(* Logix 5000 project; controller PBS_Perfusion vendor 1 type 14 code 217 rev 32.14; software revision 32.03; part 10 of 27 *)
(* tags used below, declared in another part *)
   Cfg_HasOper : BOOL;   // 1=Operator (unlocked) exists, can be selected
   Cfg_HasOperLocked : BOOL;   // 1=Operator Locked exists, can be selected
   Cfg_HasProg : BOOL;   // 1=Program (unlocked) exists, can be selected
   Cfg_HasProgLocked : BOOL;   // 1=Program Locked exists, can be selected
   Cfg_HasExt : BOOL;   // 1=External exists, can be selected
   Cfg_HasMaint : BOOL;   // 1=Maintenance exists, can be selected
   Cfg_HasMOoS : BOOL;   // 1=Maintenance Out of Service exists, can be selected
   Cfg_OvrdOverLock : BOOL;   // 1=Override supersedes Prog/Oper Lock, 0=don't override Lock
   Cfg_ExtOverLock : BOOL;   // 1=External supersedes Prog/Oper Lock, 0=don't override Lock
   Cfg_ProgNormal : BOOL;   // Normal Source: 1=Program if no requests; 0=Operator if no requests
   Cfg_PCmdPriority : BOOL;   // Command Priority: 1=Program Cmds Win; 0=Operator Cmds Win
   Cfg_PCmdProgAsLevel : BOOL;   // 1=PCmd_Prog used as a Level (1=Prog, 0=Oper)
   Cfg_PCmdLockAsLevel : BOOL;   // 1=PCmd_Lock used as a Level (1=Lock, 0=Unlock)
   Cfg_ExtAcqAsLevel : BOOL;   // 1=XCmd_Acq used as Level (1=Acq, 0=Rel)
   MCmd_Acq : BOOL;   // Maintenance Command to Acquire (Oper/Prog/Ovrd to Maint)
   OCmd_Oper : BOOL;   // Operator Command to select Operator (Prog to Oper)
   OCmd_Prog : BOOL;   // Operator Command to select Program (Oper to Prog)
   OCmd_Lock : BOOL;   // Operator Command to Lock Operator (disallow Program)
   Sts_eSrc : INT;   // Selection enum: .8=Ext, .7=OoS, .6=Oper, .5=Prog, .4=Ovrd, .3=Maint, .2=Hand, .1=Norm, .0=Lock
   Sts_bSrc : INT;   // Active Selection bitmap (for HMI totem pole)
   Sts_ProgOperSel : BOOL;   // Prog/Oper selection (latch) state, 1=Program, 0=Operator
   Sts_ProgOperLock : BOOL;   // Prog/Oper lock (latch) state, 1=Locked, 0=Unlocked
   MRdy_OoS : BOOL;   // 1=Ready for MCmd_OoS (enables HMI button)
   MRdy_IS : BOOL;   // 1=Ready for MCmd_IS (enables HMI button)
   MRdy_Acq : BOOL;   // 1=Ready for MCmd_Acq (enables HMI button)
   XRdy_Acq : BOOL;   // 1=Ready for XCmd_Acq (enables HMI button)
   XRdy_Rel : BOOL;   // 1=Ready for XCmd_Rel (enables HMI button)
   ORdy_Oper : BOOL;   // 1=Ready for OCmd_Oper (enables HMI button)
   ORdy_Prog : BOOL;   // 1=Ready for OCmd_Prog (enables HMI button)
   ORdy_Lock : BOOL;   // 1=Ready for OCmd_Lock (enables HMI button)
   ORdy_Normal : BOOL;   // 1=Ready for OCmd_Normal (enables HMI button)
   P_CmdSrc : BOOL;   // Unique Parameter Name for auto - discovery
   Wrk_ProgOperSel : BOOL;   // Internal Program (1) / Operator (0) selection result
   Wrk_ProgOperLock : BOOL;   // Internal Prog/Oper Lock (1) / Unlock (0) selection result
   Wrk_Prog : BOOL;   // Internal Program (1) / Operator (0) selection progress
   Wrk_MOoS : BOOL;   // Internal Maintenance Out of Service (1) / In Service (0) latch
   Wrk_Maint : BOOL;   // Internal Maintenance Acquire (1) / Release (0) latch
   Wrk_Lock : BOOL;   // Internal Prog/Oper Lock (1) / Unlock (0) selection progress
   Wrk_Init : BOOL;   // 1=Initialized, 0=Initialization is required (e.g., powerup)
   Wrk_Ext : BOOL;   // Internal latch of External selection (1=Ext acquired)
   REAL : DINT;
(* P_CmdSrc, continued *)

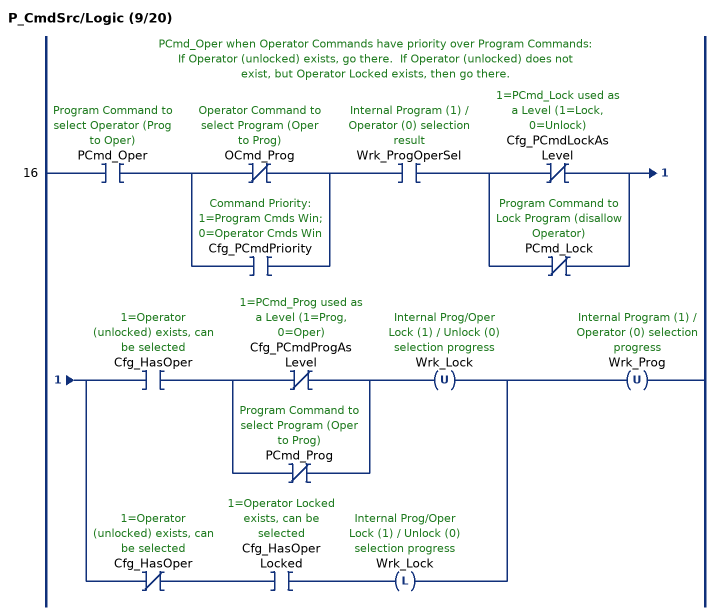
   [picture p204: P_CmdSrc/Logic rungs 16-16]
   // PCmd_Oper when Operator Commands have priority over Program Commands:
   // If Operator (unlocked) exists, go there.  If Operator (unlocked) does not
   // exist, but Operator Locked exists, then go there.
   16: XIC(PCmd_Oper)[XIO(OCmd_Prog) ,XIC(Cfg_PCmdPriority) ]XIC(Wrk_ProgOperSel)[XIO(Cfg_PCmdLockAsLevel) ,XIO(PCmd_Lock) ][XIC(Cfg_HasOper) [XIO(Cfg_PCmdProgAsLevel) ,XIO(PCmd_Prog) ] OTU(Wrk_Lock) ,XIO(Cfg_HasOper) XIC(Cfg_HasOperLocked) OTL(Wrk_Lock) ]OTU(Wrk_Prog);
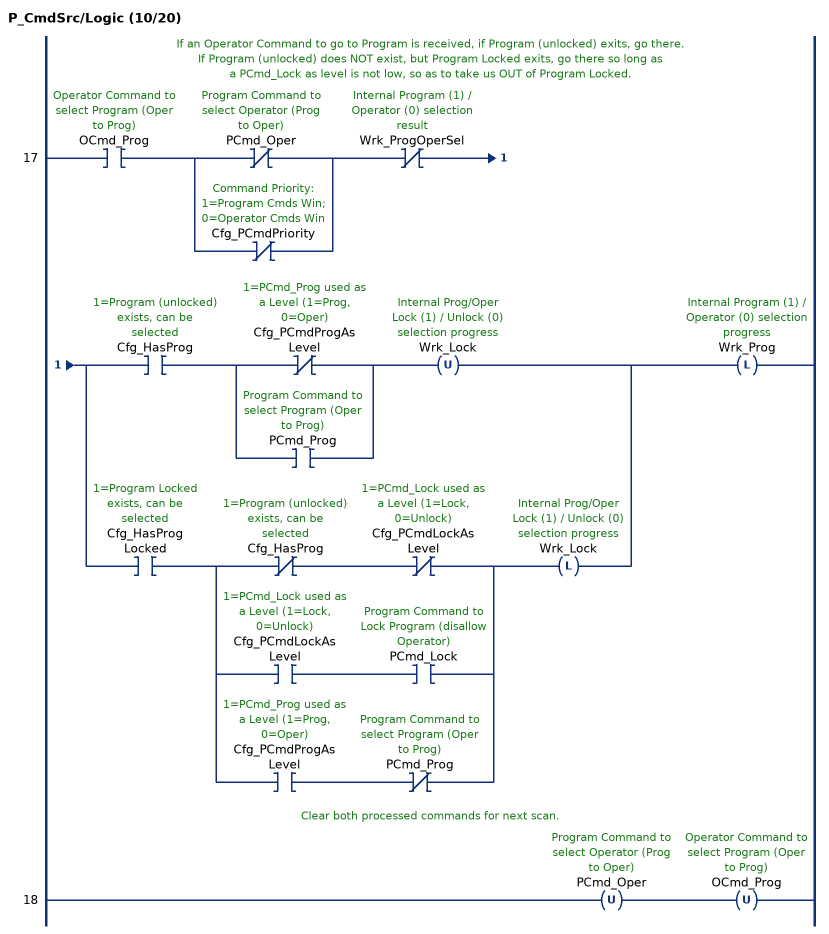
   // If an Operator Command to go to Program is received, if Program (unlocked) exits, go there.
   // If Program (unlocked) does NOT exist, but Program Locked exits, go there so long as
   // a PCmd_Lock as level is not low, so as to take us OUT of Program Locked.
   17: XIC(OCmd_Prog)[XIO(PCmd_Oper) ,XIO(Cfg_PCmdPriority) ]XIO(Wrk_ProgOperSel)[XIC(Cfg_HasProg) [XIO(Cfg_PCmdProgAsLevel) ,XIC(PCmd_Prog) ] OTU(Wrk_Lock) ,XIC(Cfg_HasProgLocked) [XIO(Cfg_HasProg) XIO(Cfg_PCmdLockAsLevel) ,XIC(Cfg_PCmdLockAsLevel) XIC(PCmd_Lock) ,XIC(Cfg_PCmdProgAsLevel) XIO(PCmd_Prog) ] OTL(Wrk_Lock) ]OTL(Wrk_Prog);
   // Clear both processed commands for next scan.
   18: OTU(PCmd_Oper)OTU(OCmd_Prog);
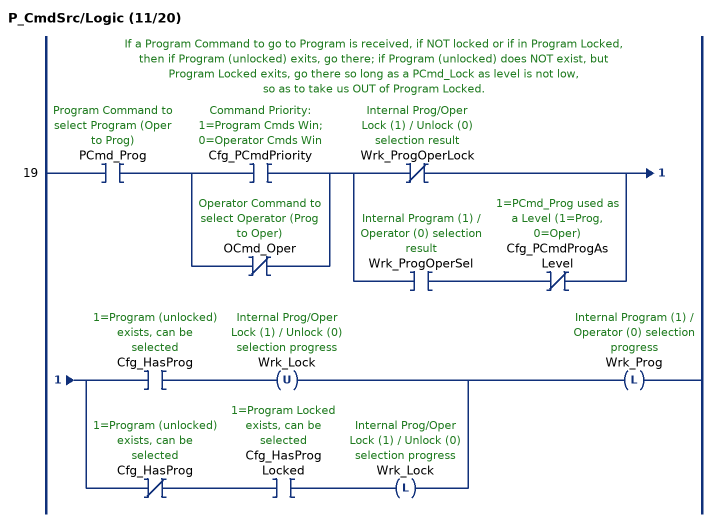
   // If a Program Command to go to Program is received, if NOT locked or if in Program Locked,
   // then if Program (unlocked) exits, go there; if Program (unlocked) does NOT exist, but
   // Program Locked exits, go there so long as a PCmd_Lock as level is not low,
   // so as to take us OUT of Program Locked.
   19: XIC(PCmd_Prog)[XIC(Cfg_PCmdPriority) ,XIO(OCmd_Oper) ][XIO(Wrk_ProgOperLock) ,XIC(Wrk_ProgOperSel) XIO(Cfg_PCmdProgAsLevel) ][XIC(Cfg_HasProg) OTU(Wrk_Lock) ,XIO(Cfg_HasProg) XIC(Cfg_HasProgLocked) OTL(Wrk_Lock) ]OTL(Wrk_Prog);
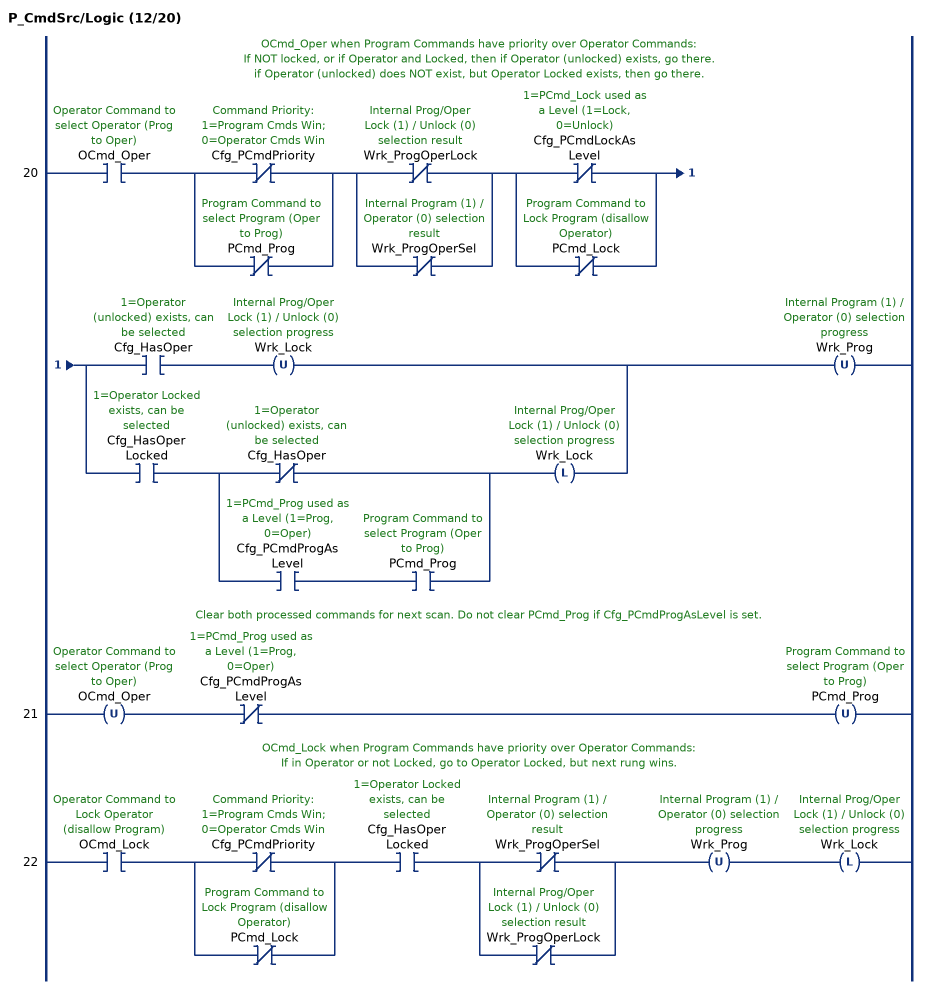
   // OCmd_Oper when Program Commands have priority over Operator Commands:
   // If NOT locked, or if Operator and Locked, then if Operator (unlocked) exists, go there.
   // if Operator (unlocked) does NOT exist, but Operator Locked exists, then go there.
   20: XIC(OCmd_Oper)[XIO(Cfg_PCmdPriority) ,XIO(PCmd_Prog) ][XIO(Wrk_ProgOperLock) ,XIO(Wrk_ProgOperSel) ][XIO(Cfg_PCmdLockAsLevel) ,XIO(PCmd_Lock) ][XIC(Cfg_HasOper) OTU(Wrk_Lock) ,XIC(Cfg_HasOperLocked) [XIO(Cfg_HasOper) ,XIC(Cfg_PCmdProgAsLevel) XIC(PCmd_Prog) ] OTL(Wrk_Lock) ]OTU(Wrk_Prog);
   // Clear both processed commands for next scan. Do not clear PCmd_Prog if Cfg_PCmdProgAsLevel is set.
   21: OTU(OCmd_Oper)XIO(Cfg_PCmdProgAsLevel)OTU(PCmd_Prog);
   // OCmd_Lock when Program Commands have priority over Operator Commands:
   // If in Operator or not Locked, go to Operator Locked, but next rung wins.
   22: XIC(OCmd_Lock)[XIO(Cfg_PCmdPriority) ,XIO(PCmd_Lock) ]XIC(Cfg_HasOperLocked)[XIO(Wrk_ProgOperSel) ,XIO(Wrk_ProgOperLock) ]OTU(Wrk_Prog)OTL(Wrk_Lock);
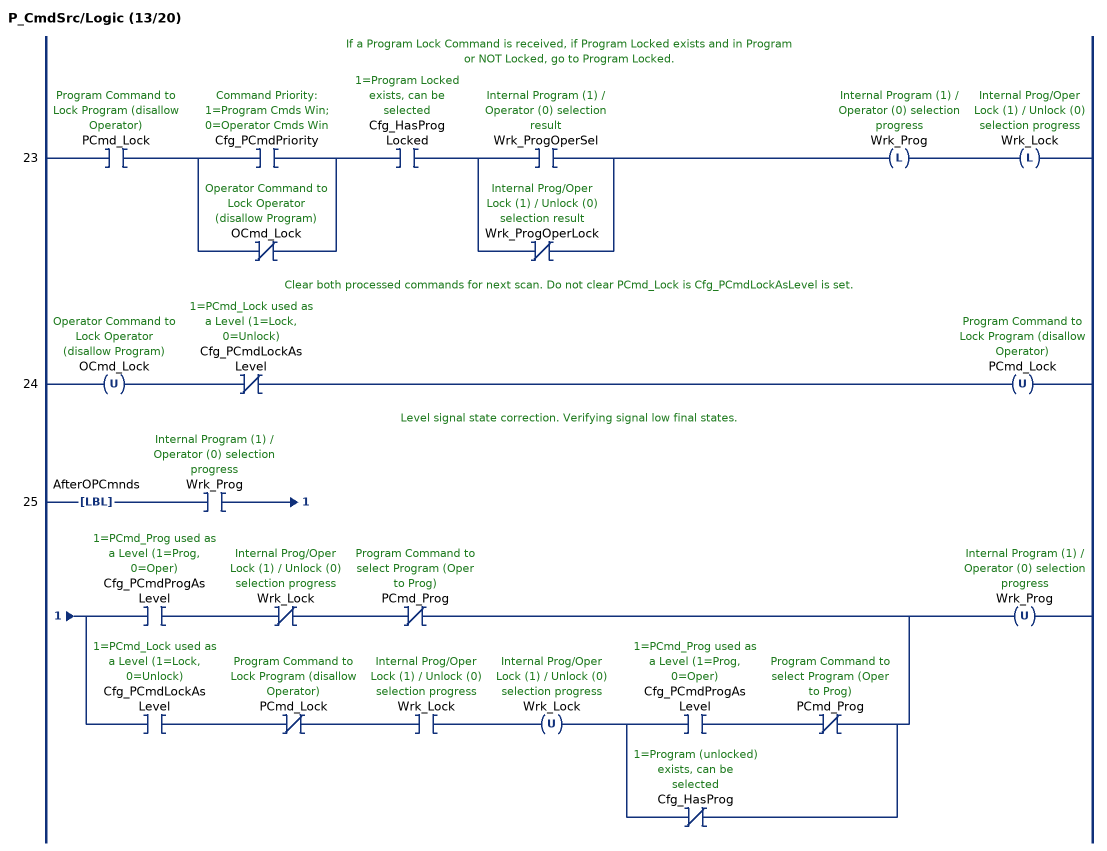
   // If a Program Lock Command is received, if Program Locked exists and in Program
   // or NOT Locked, go to Program Locked.
   23: XIC(PCmd_Lock)[XIC(Cfg_PCmdPriority) ,XIO(OCmd_Lock) ]XIC(Cfg_HasProgLocked)[XIC(Wrk_ProgOperSel) ,XIO(Wrk_ProgOperLock) ]OTL(Wrk_Prog)OTL(Wrk_Lock);
   // Clear both processed commands for next scan. Do not clear PCmd_Lock is Cfg_PCmdLockAsLevel is set.
   24: OTU(OCmd_Lock)XIO(Cfg_PCmdLockAsLevel)OTU(PCmd_Lock);
   // Level signal state correction. Verifying signal low final states.
   25: LBL(AfterOPCmnds)XIC(Wrk_Prog)[XIC(Cfg_PCmdProgAsLevel) XIO(Wrk_Lock) XIO(PCmd_Prog) ,XIC(Cfg_PCmdLockAsLevel) XIO(PCmd_Lock) XIC(Wrk_Lock) OTU(Wrk_Lock) [XIC(Cfg_PCmdProgAsLevel) XIO(PCmd_Prog) ,XIO(Cfg_HasProg) ] ]OTU(Wrk_Prog);
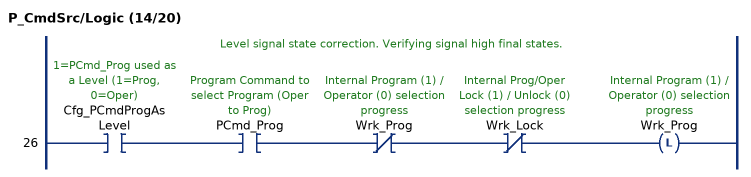
   // Level signal state correction. Verifying signal high final states.
   26: XIC(Cfg_PCmdProgAsLevel)XIC(PCmd_Prog)XIO(Wrk_Prog)XIO(Wrk_Lock)OTL(Wrk_Prog);
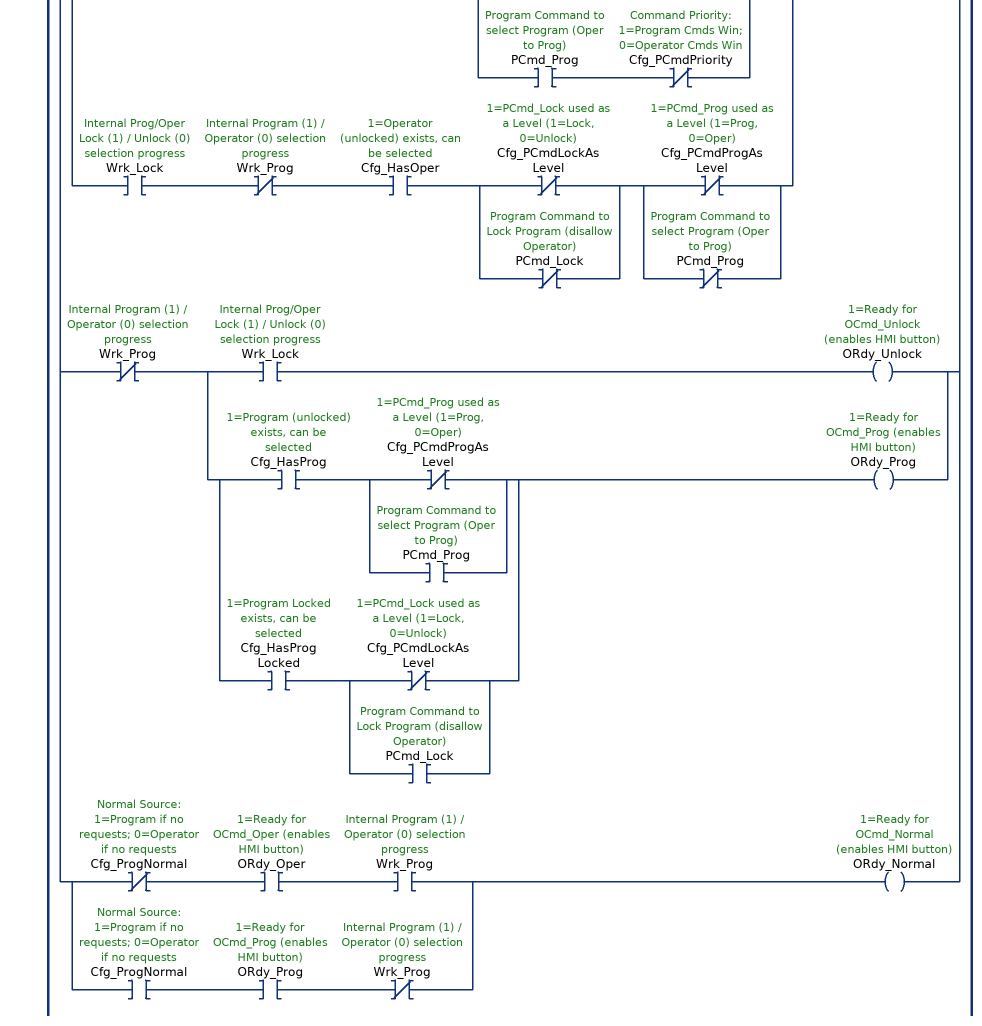
   // ============================================================
   // MAINTENANCE AND OPERATOR COMMAND READIES
   // ============================================================
   // This rung generates the "ORdy_" and "MRdy_" bits that signify to the
   // HMI that the corresponding command should "do" something
   // and the command button should be enabled on the display.
   // NOTE ON MAINTENANCE ACQUIRE: Ready for MCmd_Acq if Maintenance
   // is allowed and the internal Maintenance latch is NOT set.  However,
   // we need to display Ready even if latch IS set so that Sts_MAcqRcvd
   // can blink to reset an external Maintenance expiration timer!!!
   // #####  V4.10.00  2019-03-08:  Added XRdy_Acq, XRdy_Rel so External Acq/Rel can be used on HMI .  #####
   27: [XIC(Cfg_HasMaint) [OTE(MRdy_Acq) ,XIC(Wrk_Maint) OTE(MRdy_Rel) ] ,XIC(Cfg_HasMOoS) [XIC(Wrk_MOoS) OTE(MRdy_IS) ,XIO(Wrk_MOoS) OTE(MRdy_OoS) ] ,XIC(Cfg_HasExt) XIO(Cfg_ExtAcqAsLevel) [XIC(Wrk_Ext) OTE(XRdy_Rel) ,XIO(Wrk_Ext) XIO(Inp_ExtInh) OTE(XRdy_Acq) ] ,XIO(Wrk_Lock) XIC(Cfg_HasOperLocked) OTE(ORdy_Lock) ,[XIO(Wrk_Lock) XIC(Wrk_Prog) [XIC(Cfg_HasOper) XIO(Cfg_PCmdProgAsLevel) ,XIC(Cfg_HasOperLocked) [XIO(Cfg_PCmdProgAsLevel) ,XIC(PCmd_Prog) XIO(Cfg_PCmdPriority) ] ] ,XIC(Wrk_Lock) XIO(Wrk_Prog) XIC(Cfg_HasOper) [XIO(Cfg_PCmdLockAsLevel) ,XIO(PCmd_Lock) ] [XIO(Cfg_PCmdProgAsLevel) ,XIO(PCmd_Prog) ] ] OTE(ORdy_Oper) ,XIO(Wrk_Prog) [XIC(Wrk_Lock) OTE(ORdy_Unlock) ,[XIC(Cfg_HasProg) [XIO(Cfg_PCmdProgAsLevel) ,XIC(PCmd_Prog) ] ,XIC(Cfg_HasProgLocked) [XIO(Cfg_PCmdLockAsLevel) ,XIC(PCmd_Lock) ] ] OTE(ORdy_Prog) ] ,[XIO(Cfg_ProgNormal) XIC(ORdy_Oper) XIC(Wrk_Prog) ,XIC(Cfg_ProgNormal) XIC(ORdy_Prog) XIO(Wrk_Prog) ] OTE(ORdy_Normal) ];
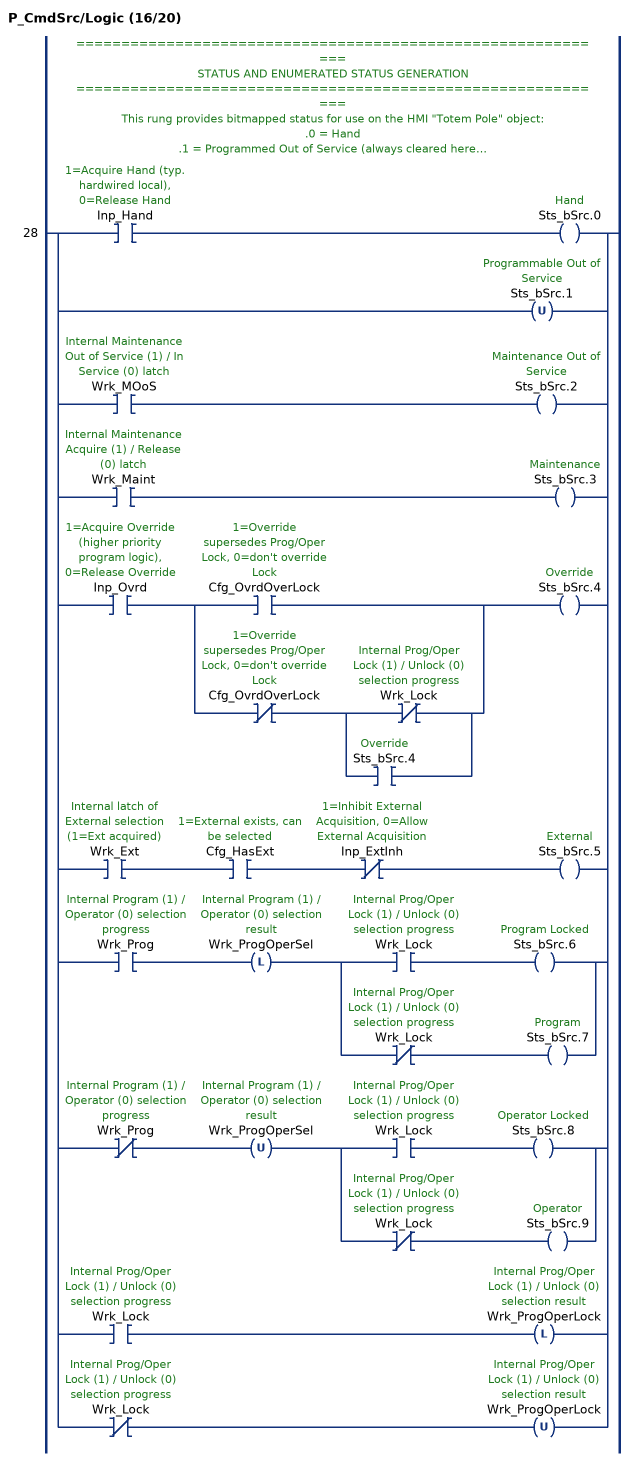
   // ============================================================
   // STATUS AND ENUMERATED STATUS GENERATION
   // ============================================================
   // This rung provides bitmapped status for use on the HMI "Totem Pole" object:
   // .0 = Hand
   // .1 = Programmed Out of Service (always cleared here)
   // .2 = Maintenance Out of Service
   // .3 = Maintenance
   // .4= Override
   // .5 = External
   // .6 = Program Locked
   // .7 = Program
   // .8 = Operator Locked
   // .9 = Operator
   // In addition, the final selections of the Program / Operator selection latch
   // and the Prog/Oper lock latch are captured for use next scan.
   // #####  V4.10.00  2019-03-08:  Added XCmd_Acq, XCmd_Rel, Cfg_ExtAcqAsLevel, removed Inp_Ext.  #####
   28: [XIC(Inp_Hand) OTE(Sts_bSrc.0) ,OTU(Sts_bSrc.1) ,XIC(Wrk_MOoS) OTE(Sts_bSrc.2) ,XIC(Wrk_Maint) OTE(Sts_bSrc.3) ,XIC(Inp_Ovrd) [XIC(Cfg_OvrdOverLock) ,XIO(Cfg_OvrdOverLock) [XIO(Wrk_Lock) ,XIC(Sts_bSrc.4) ] ] OTE(Sts_bSrc.4) ,XIC(Wrk_Ext) XIC(Cfg_HasExt) XIO(Inp_ExtInh) OTE(Sts_bSrc.5) ,XIC(Wrk_Prog) OTL(Wrk_ProgOperSel) [XIC(Wrk_Lock) OTE(Sts_bSrc.6) ,XIO(Wrk_Lock) OTE(Sts_bSrc.7) ] ,XIO(Wrk_Prog) OTU(Wrk_ProgOperSel) [XIC(Wrk_Lock) OTE(Sts_bSrc.8) ,XIO(Wrk_Lock) OTE(Sts_bSrc.9) ] ,XIC(Wrk_Lock) OTL(Wrk_ProgOperLock) ,XIO(Wrk_Lock) OTU(Wrk_ProgOperLock) ];
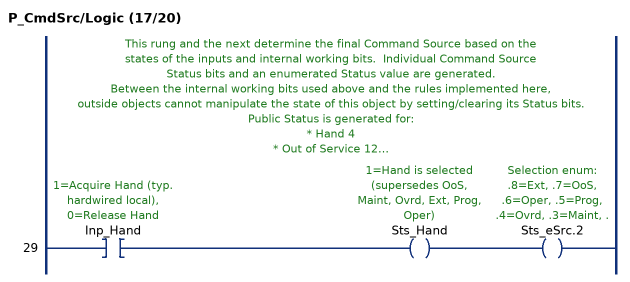
   // This rung and the next determine the final Command Source based on the
   // states of the inputs and internal working bits.  Individual Command Source
   // Status bits and an enumerated Status value are generated.
   // Between the internal working bits used above and the rules implemented here,
   // outside objects cannot manipulate the state of this object by setting/clearing its Status bits.
   // Public Status is generated for:
   // * Hand 4
   // * Out of Service 129
   // * Maintenance 8
   // * Override 16
   // * External 256
   // * Program 32
   // * Operator 64
   // * Program / Operator Lock status 33/65
   // * Command Source = Normal 34/66
   29: XIC(Inp_Hand)OTE(Sts_Hand)OTE(Sts_eSrc.2);
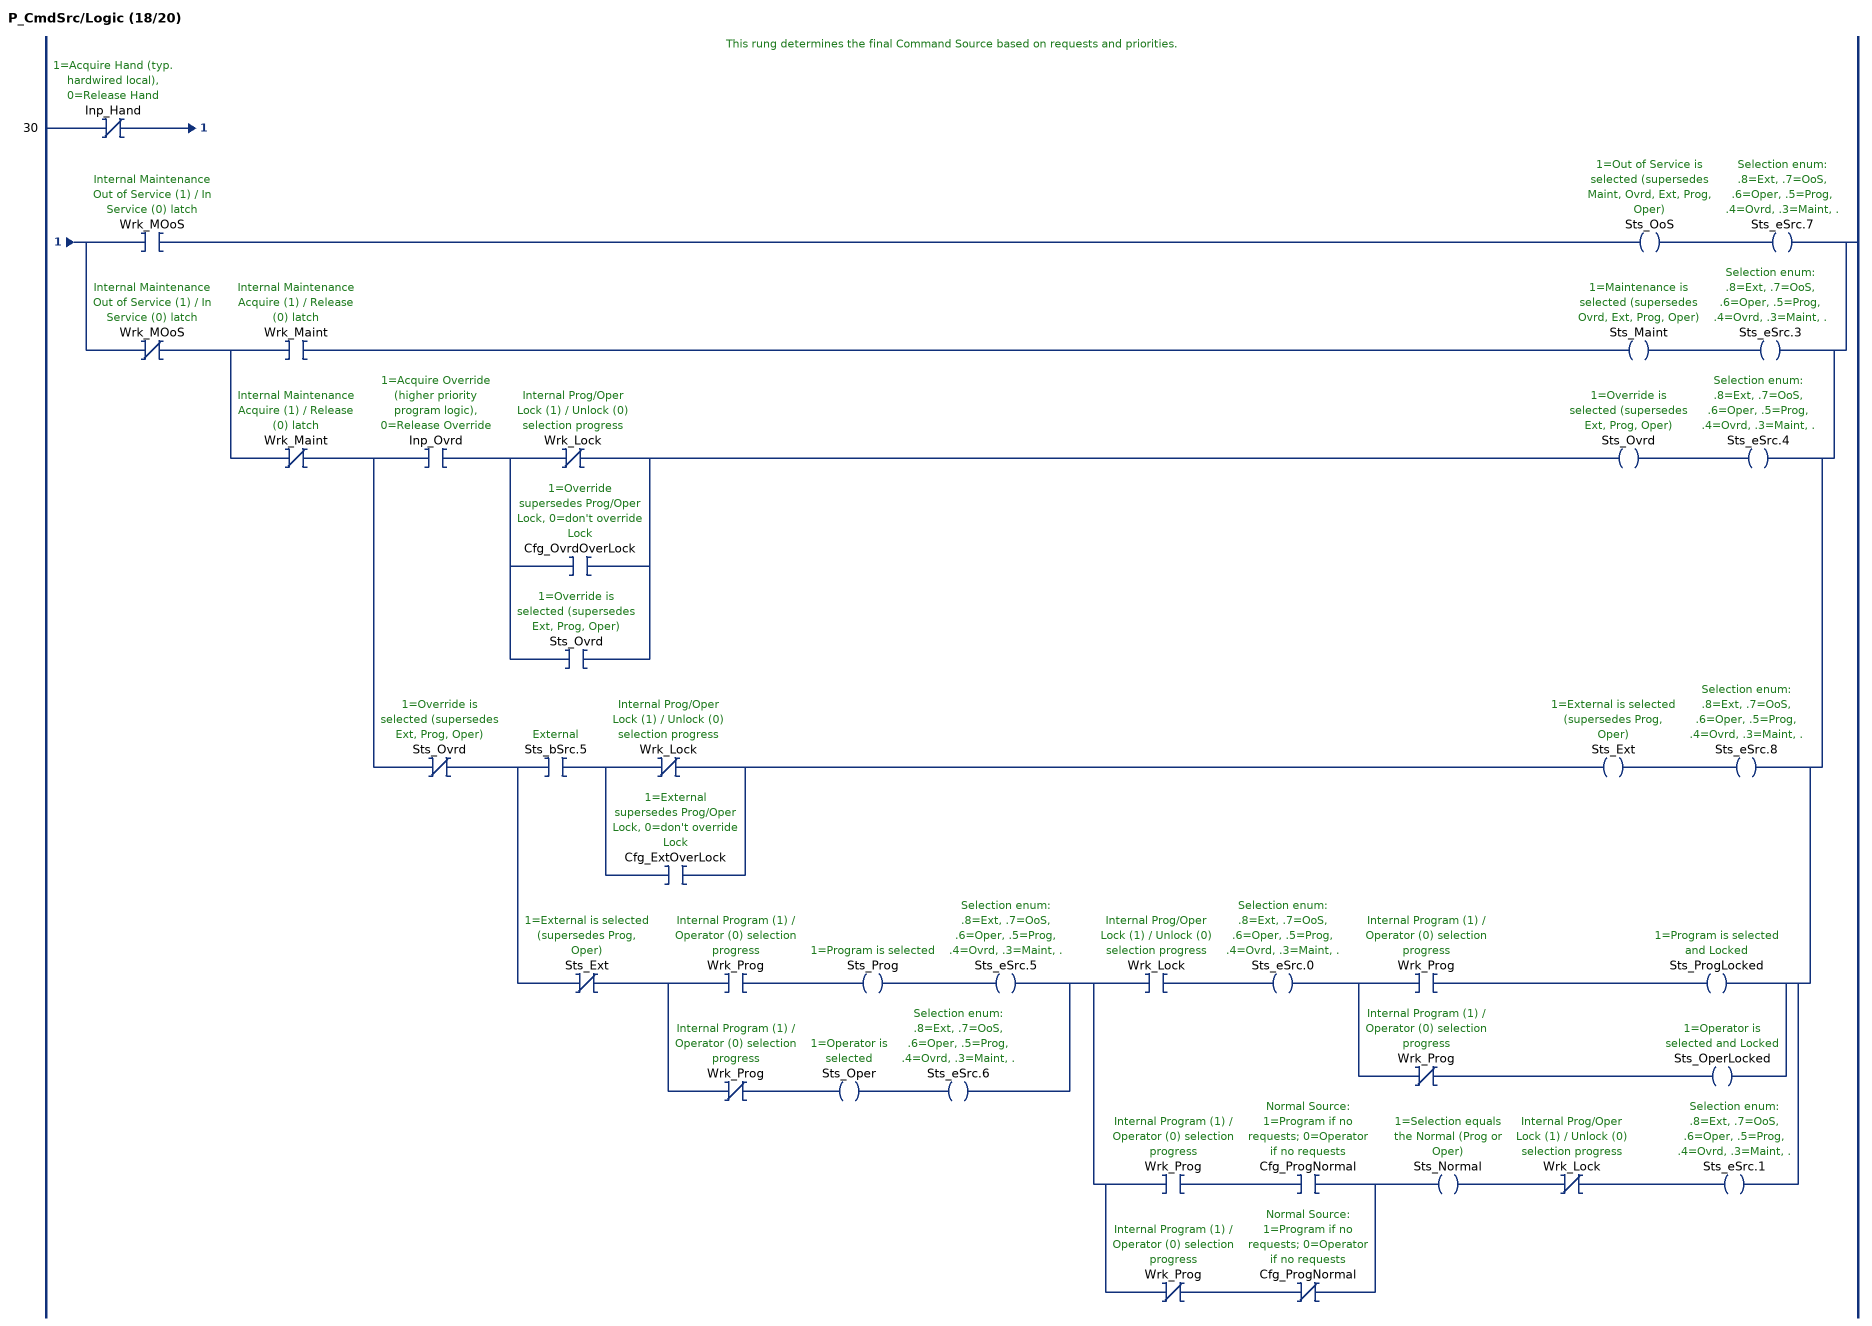
   // This rung determines the final Command Source based on requests and priorities.
   30: XIO(Inp_Hand)[XIC(Wrk_MOoS) OTE(Sts_OoS) OTE(Sts_eSrc.7) ,XIO(Wrk_MOoS) [XIC(Wrk_Maint) OTE(Sts_Maint) OTE(Sts_eSrc.3) ,XIO(Wrk_Maint) [XIC(Inp_Ovrd) [XIO(Wrk_Lock) ,XIC(Cfg_OvrdOverLock) ,XIC(Sts_Ovrd) ] OTE(Sts_Ovrd) OTE(Sts_eSrc.4) ,XIO(Sts_Ovrd) [XIC(Sts_bSrc.5) [XIO(Wrk_Lock) ,XIC(Cfg_ExtOverLock) ] OTE(Sts_Ext) OTE(Sts_eSrc.8) ,XIO(Sts_Ext) [XIC(Wrk_Prog) OTE(Sts_Prog) OTE(Sts_eSrc.5) ,XIO(Wrk_Prog) OTE(Sts_Oper) OTE(Sts_eSrc.6) ] [XIC(Wrk_Lock) OTE(Sts_eSrc.0) [XIC(Wrk_Prog) OTE(Sts_ProgLocked) ,XIO(Wrk_Prog) OTE(Sts_OperLocked) ] ,[XIC(Wrk_Prog) XIC(Cfg_ProgNormal) ,XIO(Wrk_Prog) XIO(Cfg_ProgNormal) ] OTE(Sts_Normal) XIO(Wrk_Lock) OTE(Sts_eSrc.1) ] ] ] ] ];
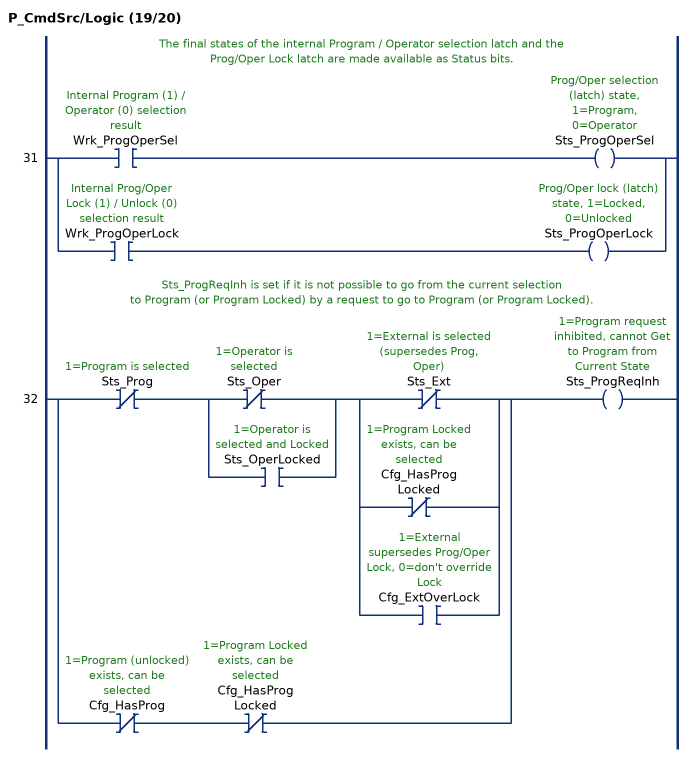
   // The final states of the internal Program / Operator selection latch and the
   // Prog/Oper Lock latch are made available as Status bits.
   31: [XIC(Wrk_ProgOperSel) OTE(Sts_ProgOperSel) ,XIC(Wrk_ProgOperLock) OTE(Sts_ProgOperLock) ];
   // Sts_ProgReqInh is set if it is not possible to go from the current selection
   // to Program (or Program Locked) by a request to go to Program (or Program Locked).
   32: [XIO(Sts_Prog) [XIO(Sts_Oper) ,XIC(Sts_OperLocked) ] [XIO(Sts_Ext) ,XIO(Cfg_HasProgLocked) ,XIC(Cfg_ExtOverLock) ] ,XIO(Cfg_HasProg) XIO(Cfg_HasProgLocked) ]OTE(Sts_ProgReqInh);
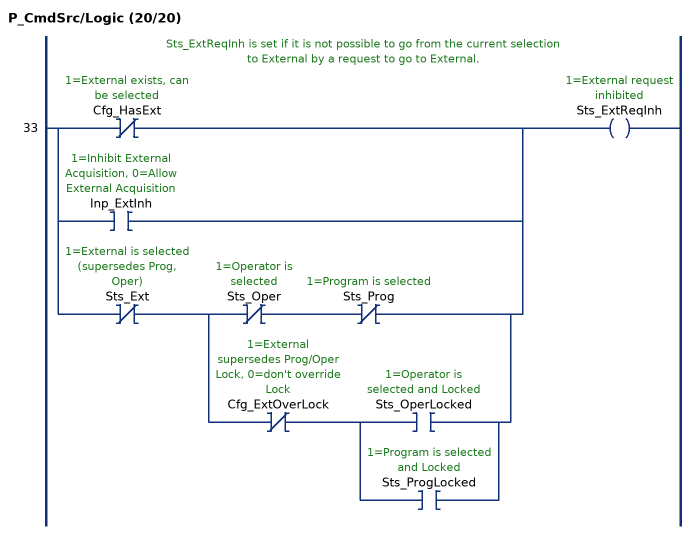
   // Sts_ExtReqInh is set if it is not possible to go from the current selection
   // to External by a request to go to External.
   33: [XIO(Cfg_HasExt) ,XIC(Inp_ExtInh) ,XIO(Sts_Ext) [XIO(Sts_Oper) XIO(Sts_Prog) ,XIO(Cfg_ExtOverLock) [XIC(Sts_OperLocked) ,XIC(Sts_ProgLocked) ] ] ]OTE(Sts_ExtReqInh);
END_ROUTINE

ROUTINE Prescan   (* ladder *)
// Sets internal state and enumerated / bit status to "not initialized".
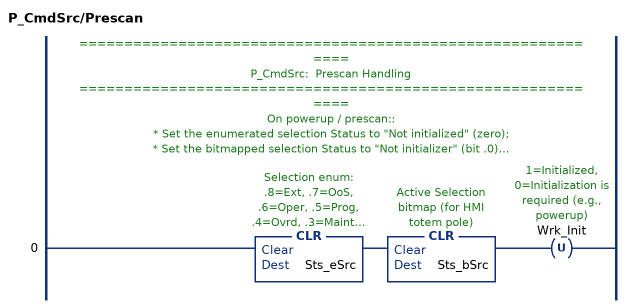
   // ============================================================
   // P_CmdSrc:  Prescan Handling
   // ============================================================
   // On powerup / prescan::
   // * Set the enumerated selection Status to "Not initialized" (zero);
   // * Set the bitmapped selection Status to "Not initializer" (bit .0);
   // * Flag the instruction to execute the initialization rungs when run.
   0: CLR(Sts_eSrc)CLR(Sts_bSrc)OTU(Wrk_Init);
END_ROUTINE
END_ADD_ON_INSTRUCTION

ADD_ON_INSTRUCTION P_D4SD   (* revision 4.10 .01 Release, vendor Rockwell Automation, ExecutePrescan, ExecuteEnableInFalse *)
// 2-, 3- or 4-State Device
// Revision note:
// See Instruction Help for a summary of changes, and see 4.10 Release Notes for details.
// Help:
// Copyright © Rockwell Automation, Inc.  All Rights Reserved.
// This Instruction controls and monitors feedback from a Discrete 2-State,
// 3-State or 4-State Device, and provides:
//   *  Operator and Program Commands to select one of the 2, 3 or 4 states
//   *  User-configurable text labels for the states
//   *  Per-State setting, clearing or holding of four user-configurable outputs
//   *  Per-State monitoring of four feedbacks (on, off or don't care) to confirm state
//   *  Detection of failure to reach the target state (when feedbacks are used)
//   *  Monitoring of Permissive conditions to allow commanding to each state
//   *  Monitoring of Interlock conditions to return device to State 0
//   *  Operation in Hand, Maintenance, Override, Program and Operator Modes
//   *  Simulation, providing feedback of a working device while disabling output
//        (keeping de-energized)
//   *  Monitoring of I/O communication status
//   *  Alarms for Fail to reach target state (if feedbacks are used), Device Failure
//       (reported by device using an input), Interlock Trip, I/O Fault
//   *  "Available" status for use by automation logic to know whether the
//       device can be controlled by other objects.
// Command Sources are arbitrated by a P_CmdSrc Add-On Instruction instance.
// Command Sources: Operator, Program, External, Override, Maintenance, Out of
// Service, Hand.  Alarms are provided by P_Alarm Add-On Instruction instances.
// SUMMARY OF CHANGES FROM PREVIOUS VERSION (4.10.00)
// See 4.10 Release Notes for details.
// * No changes, uprevved because P_CmdSrc 4.10.01 is used.
// SUMMARY OF CHANGES FROM PREVIOUS VERSION (4.00.00)
// See 4.10 Release Notes for details.
// * Changed availability to use input availability from interlocks.
// * Added audible alert on commanded energize/state change.
// * Added Inp_HornInh to disable Horn operation.
// * Modified logic to correct confgurable shed action.
// * Updated to P_CmdSrc V4.10.00.
// * Added Cfg_HasMoreObj.
// SUMMARY OF CHANGES FROM PREVIOUS VERSION (3.5-11)
// See 4.00 Release Notes for details.
// * Changed Inf_ items to HMI_, and added Cfg_Area for security.
// * Added notify and unack count rollup for Channel object.
// * Changed "Mode" to "Command Source" using P_CmdSrc 4.00.00.
// * Deleted Cfg_PCmdClear; all Program Commands are now self-clearing.
// * Aligned ready bit naming with command bit names.
// * All OCmds/MCmds and ORdys/MRdys are now Local Tags.
// * Added Sts_AckReqd and Sts_ResetReqd for use by external objects.
// * Changed delay / time configuration items to REAL seconds.
VAR_INPUT
   Inp_FdbkA : BOOL; {visible}   // Input Signal: Feedback A from device
   Inp_FdbkB : BOOL; {visible}   // Input Signal: Feedback B from device
   Inp_FdbkC : BOOL; {visible}   // Input Signal: Feedback C from device
   Inp_FdbkD : BOOL; {visible}   // Input Signal: Feedback D from device
   Inp_DeviceFault : BOOL;   // Input Signal: Device Fault from device
   Inp_PermOK0 : BOOL := 1; {visible}   // 1=Permissives OK, device can be commanded to State 0
   Inp_NBPermOK0 : BOOL := 1; {visible}   // 1=Non-Bypassable Permissives OK, device can be commanded to State 0
   Inp_PermOK1 : BOOL := 1; {visible}   // 1=Permissives OK, device can be commanded to State 1
   Inp_NBPermOK1 : BOOL := 1; {visible}   // 1=Non-Bypassable Permissives OK, device can be commanded to State 1
   Inp_PermOK2 : BOOL := 1; {visible}   // 1=Permissives OK, device can be commanded to State 2
   Inp_NBPermOK2 : BOOL := 1; {visible}   // 1=Non-Bypassable Permissives OK, device can be commanded to State 2
   Inp_PermOK3 : BOOL := 1; {visible}   // 1=Permissives OK, device can be commanded to State 3
   Inp_NBPermOK3 : BOOL := 1; {visible}   // 1=Non-Bypassable Permissives OK, device can be commanded to State 3
   Inp_IntlkOK : BOOL := 1; {visible}   // 1=Interlocks OK, 0=Not OK, go to State 0
   Inp_NBIntlkOK : BOOL := 1; {visible}   // 1=Non-Bypassable Interlocks OK, 0=Not OK, go to State 0
   Inp_IntlkAvail : BOOL;   // 1 = Interlock Availibility OK
   Inp_IOFault : BOOL;   // Input Communication Status 0=OK, 1=fail
   Inp_Sim : BOOL;   // 1=Simulate working device; 0=Control actual device
   Inp_Hand : ALIAS FOR CmdSrc.Inp_Hand;
   Inp_Ovrd : ALIAS FOR CmdSrc.Inp_Ovrd;
   Inp_OvrdCmd : DINT;   // Override Device Command: 0=None, 1=St.0, 2=St.1, 3=St.2, 4=St.3
   Inp_ExtInh : ALIAS FOR CmdSrc.Inp_ExtInh;
   Inp_HornInh : BOOL;   // 1 = Inhibit audible alert, 0 = Alllow audible alert
   Inp_Reset : BOOL;   // 1=Reset all fault conditions and latched Alarms
   Cfg_St0onShed : BOOL;   // 1=Go to State 0 on Shed, 0=Hold position on Shed
   Cfg_NumStates : DINT := 2;   // Number of device states (2..4)
   Cfg_OutSt0Write : SINT := 2#0000_1111;   // Bit=1: write output in state 0, Bit=0: leave in last state
   Cfg_OutSt0State : SINT := 2#0000_0001;   // (if written) Bit=1: output set in State 0, Bit=0: output cleared
   Cfg_OutSt1Write : SINT := 2#0000_1111;   // Bit=1: write output in state 1, Bit=0: leave in last state
   Cfg_OutSt1State : SINT := 2#0000_0010;   // (if written) Bit=1: output set in State 1, Bit=0: output cleared
   Cfg_OutSt2Write : SINT := 2#0000_1111;   // Bit=1: write output in state 2, Bit=0: leave in last state
   Cfg_OutSt2State : SINT := 2#0000_0100;   // (if written) Bit=1: output set in State 2, Bit=0: output cleared
   Cfg_OutSt3Write : SINT := 2#0000_1111;   // Bit=1: write output in state 3, Bit=0: leave in last state
   Cfg_OutSt3State : SINT := 2#0000_1000;   // (if written) Bit=1: output set in State 3, Bit=0: output cleared
   Cfg_FdbkSt0Check : SINT;   // Bit=1: Check Feedback in state 0, Bit=0: don't care
   Cfg_FdbkSt0State : SINT := 2#0000_0001;   // (if checking) Bit=1: Feedback is 1 in State 0, Bit=0: Feedback is 0
   Cfg_FdbkSt1Check : SINT;   // Bit=1: Check Feedback in state 1, Bit=0: don't care
   Cfg_FdbkSt1State : SINT := 2#0000_0010;   // (if checking) Bit=1: Feedback is 1 in State 1, Bit=0: Feedback is 0
   Cfg_FdbkSt2Check : SINT;   // Bit=1: Check Feedback in state 2, Bit=0: don't care
   Cfg_FdbkSt2State : SINT := 2#0000_0100;   // (if checking) Bit=1: Feedback is 1 in State 2, Bit=0: Feedback is 0
   Cfg_FdbkSt3Check : SINT;   // Bit=1: Check Feedback in state 3, Bit=0: don't care
   Cfg_FdbkSt3State : SINT := 2#0000_1000;   // (if checking) Bit=1: Feedback is 1 in State 3, Bit=0: Feedback is 0
   Cfg_HasPerm0Obj : BOOL;   // 1=Tells HMI a P_Perm is connected to Inp_PermOK0
   Cfg_HasPerm1Obj : BOOL;   // 1=Tells HMI a P_Perm is connected to Inp_PermOK1
   Cfg_HasPerm2Obj : BOOL;   // 1=Tells HMI a P_Perm is connected to Inp_PermOK2
   Cfg_HasPerm3Obj : BOOL;   // 1=Tells HMI a P_Perm is connected to Inp_PermOK3
   Cfg_HasIntlkObj : BOOL;   // 1=Tells HMI a P_Intlk is connected to Inp_IntlkOK
   Cfg_HasMoreObj : BOOL;   // 1=Tells HMI an object with more info is available
   Cfg_OperSt0Prio : BOOL;   // 1=OCmd_St0 any time, 0=OCmd_St0 only when Oper selected
   Cfg_ExtSt0Prio : BOOL;   // 1=XCmd_St0 any time, 0=XCmd_St0 only when Ext selected
   Cfg_OCmdResets : BOOL;   // 1=New device OCmd resets shed latches and cleared alarms, 0=OCmdReset req'd.
   Cfg_XCmdResets : BOOL;   // 1=New device XCmd resets shed latches and cleared alarms, 0=XCmdReset req'd.
   Cfg_OvrdPermIntlk : BOOL;   // 1=Override ignores Bypassable Perm/ Intlk; 0=always use Perm/Intlk
   Cfg_ShedOnFail : BOOL;   // 1=Go to State 0 and Alarm on Fail to reach position; 0=Alarm only on Fail
   Cfg_ShedOnDeviceFault : BOOL;   // 1=Go to State 0 and Alarm on Device Fault; 0=Alarm only on Device Fault
   Cfg_ShedOnIOFault : BOOL;   // 1=Go to State 0 and Alarm on I/O Fault; 0=Alarm only on I/O Fault
   Cfg_HasFailAlm : ALIAS FOR Fail.Cfg_Exists;   // 1=Fail to reach state Alarm exists and will be checked
   Cfg_HasDeviceFaultAlm : ALIAS FOR DeviceFault.Cfg_Exists;   // 1=Device Fault Alarm exists and will be checked
   Cfg_HasIntlkTripAlm : ALIAS FOR IntlkTrip.Cfg_Exists;   // 1=Interlock Trip Alarm exists and will be checked
   Cfg_HasIOFaultAlm : ALIAS FOR IOFault.Cfg_Exists;   // 1=I/O Fault Alarm exists and will be checked
   Cfg_HornOnChange : BOOL;   // 0 = Horn on energize only, 1 = Horn on any state change
   Cfg_FailResetReqd : ALIAS FOR Fail.Cfg_ResetReqd;   // 1=Reset required to clear Fail to reach state Alarm
   Cfg_DeviceFaultResetReqd : ALIAS FOR DeviceFault.Cfg_ResetReqd;   // 1=Reset required to clear Device Fault Alarm
   Cfg_IntlkTripResetReqd : ALIAS FOR IntlkTrip.Cfg_ResetReqd;   // 1=Reset required to clear Interlock Trip Alarm
   Cfg_IOFaultResetReqd : ALIAS FOR IOFault.Cfg_ResetReqd;   // 1=Reset required to clear I/O Fault Alarm
   Cfg_FailAckReqd : ALIAS FOR Fail.Cfg_AckReqd;   // 1=Acknowledge required for Fail to reach state Alarm
   Cfg_DeviceFaultAckReqd : ALIAS FOR DeviceFault.Cfg_AckReqd;   // 1=Acknowledge required for Device Fault Alarm
   Cfg_IntlkTripAckReqd : ALIAS FOR IntlkTrip.Cfg_AckReqd;   // 1=Acknowledge required for Interlock Trip Alarm
   Cfg_IOFaultAckReqd : ALIAS FOR IOFault.Cfg_AckReqd;   // 1=Acknowledge required for I/O Fault Alarm
   Cfg_FailSeverity : ALIAS FOR Fail.Cfg_Severity;   // Fail to reach state Alarm Severity: 1..250=Low, 251..500=Medium, 501..750=High, 751..1000=Urgent
   Cfg_DeviceFaultSeverity : ALIAS FOR DeviceFault.Cfg_Severity;   // Device Fault Alarm Severity: 1..250=Low, 251..500=Medium, 501..750=High, 751..1000=Urgent
   Cfg_IntlkTripSeverity : ALIAS FOR IntlkTrip.Cfg_Severity;   // Interlock Trip Alarm Severity: 1..250=Low, 251..500=Medium, 501..750=High, 751..1000=Urgent
   Cfg_IOFaultSeverity : ALIAS FOR IOFault.Cfg_Severity;   // I/O Fault Alarm Severity: 1..250=Low, 251..500=Medium, 501..750=High, 751..1000=Urgent
   Cfg_OutAPulseT : REAL;   // Time to pulse Output A (sec) (0=output held continuously)
   Cfg_OutBPulseT : REAL;   // Time to pulse Output B (sec) (0=output held continuously)
   Cfg_OutCPulseT : REAL;   // Time to pulse Output C (sec) (0=output held continuously)
   Cfg_OutDPulseT : REAL;   // Time to pulse Output D (sec) (0=output held continuously)
   Cfg_SimFdbkT : REAL := 2.0;   // Delay to echo back reaching state when in Simulation (sec)
   Cfg_StartHornT : REAL;   // Time to sound audible on commanded start (sec) (0=disabled)
   Cfg_FailT : REAL := 10.0;   // Time after new state requested to reach that state before Fault (sec)
   PSet_Owner : DINT;   // Program Owner Request ID (non-zero) or Release (zero)
   PCmd_St0 : BOOL;   // Program Command to set device to State 0
   PCmd_St1 : BOOL;   // Program Command to set device to State 1
   PCmd_St2 : BOOL;   // Program Command to set device to State 2
   PCmd_St3 : BOOL;   // Program Command to set device to State 3
   PCmd_Prog : ALIAS FOR CmdSrc.PCmd_Prog;
   PCmd_Oper : ALIAS FOR CmdSrc.PCmd_Oper;
   PCmd_Lock : ALIAS FOR CmdSrc.PCmd_Lock;
   PCmd_Unlock : ALIAS FOR CmdSrc.PCmd_Unlock;
   PCmd_Normal : ALIAS FOR CmdSrc.PCmd_Normal;
   PCmd_Reset : BOOL;   // Program Command to ResetShed Latches and Cleared Alarms
   PCmd_FailAck : ALIAS FOR Fail.PCmd_Ack;   // Program Command to Acknowledge Fail to Reach Target Position Alarm
   PCmd_FailSuppress : ALIAS FOR Fail.PCmd_Suppress;   // Program Command to Suppress Fail to Reach Target Position Alarm
   PCmd_FailUnsuppress : ALIAS FOR Fail.PCmd_Unsuppress;   // Program Command to Unsuppress Fail to Reach Target Position Alarm
   PCmd_FailUnshelve : ALIAS FOR Fail.PCmd_Unshelve;   // Program Command to Unshelve Fail to Reach Target Position Alarm
   PCmd_DeviceFaultAck : ALIAS FOR DeviceFault.PCmd_Ack;   // Program Command to Acknowledge Device Fault Alarm
   PCmd_DeviceFaultSuppress : ALIAS FOR DeviceFault.PCmd_Suppress;   // Program Command to Suppress Device Fault Alarm
   PCmd_DeviceFaultUnsuppress : ALIAS FOR DeviceFault.PCmd_Unsuppress;   // Program Command to Unsuppress Device Fault Alarm
   PCmd_DeviceFaultUnshelve : ALIAS FOR DeviceFault.PCmd_Unshelve;   // Program Command to Unshelve Device Fault Alarm
   PCmd_IntlkTripAck : ALIAS FOR IntlkTrip.PCmd_Ack;   // Program Command to Acknowledge Interlock Trip Alarm
   PCmd_IntlkTripSuppress : ALIAS FOR IntlkTrip.PCmd_Suppress;   // Program Command to Suppress Interlock Trip Alarm
   PCmd_IntlkTripUnsuppress : ALIAS FOR IntlkTrip.PCmd_Unsuppress;   // Program Command to Unsuppress Interlock Trip Alarm
   PCmd_IntlkTripUnshelve : ALIAS FOR IntlkTrip.PCmd_Unshelve;   // Program Command to Unshelve Interlock Trip Alarm
   PCmd_IOFaultAck : ALIAS FOR IOFault.PCmd_Ack;   // Program Command to Acknowledge I/O Fault Alarm
   PCmd_IOFaultSuppress : ALIAS FOR IOFault.PCmd_Suppress;   // Program Command to Suppress I/O Fault Alarm
   PCmd_IOFaultUnsuppress : ALIAS FOR IOFault.PCmd_Unsuppress;   // Program Command to Unsuppress I/O Fault Alarm
   PCmd_IOFaultUnshelve : ALIAS FOR IOFault.PCmd_Unshelve;   // Program Command to Unshelve I/O Fault Alarm
   MCmd_Rel : ALIAS FOR CmdSrc.MCmd_Rel;
   OCmd_Unlock : ALIAS FOR CmdSrc.OCmd_Unlock;
   XCmd_St0 : BOOL;   // External Command to set device to State 0
   XCmd_St1 : BOOL;   // External Command to set device to State 1
   XCmd_St2 : BOOL;   // External Command to set device to State 2
   XCmd_St3 : BOOL;   // External Command to set device to State 3
   XCmd_Acq : ALIAS FOR CmdSrc.XCmd_Acq;
   XCmd_Rel : ALIAS FOR CmdSrc.XCmd_Rel;
   XCmd_Reset : BOOL;   // External Command to reset shed latches and cleared alarms
END_VAR
VAR_OUTPUT
   Out_A : BOOL; {access Read Only, visible}   // Output A to Device
   Out_B : BOOL; {access Read Only, visible}   // Output B to Device
   Out_C : BOOL; {access Read Only, visible}   // Output C to Device
   Out_D : BOOL; {access Read Only, visible}   // Output D to Device
   Out_Horn : BOOL; {access Read Only}   // 1=Sound audible prior to commanded energize/ state change
   SrcQ_IO : DINT; {access Read Only}   // Source and Quality of primary I/O (enumeration)
   SrcQ : DINT; {access Read Only}   // Source and Quality of primary Val/Sts (enumeration)
   Val_Cmd : DINT; {access Read Only}   // Device Command 0=None, 1=State 0, 2=State 1, 3=State 2, 4=State 3
   Val_Sts : DINT; {access Read Only}   // Device Confirmed Sts 0=Powerup/Reset, 1=State0, 2=State1, 3=State2, 4=State3, 9=Moving
   Val_Fault : DINT; {access Read Only}   // Device Fault Status 0=None, 16=PositionFail, 17=DeviceFault, 32=I/OFault, 34=CfgErr
   Val_NotifyAll : DINT; {access Read Only}   // Highest Alarm prio and ack status this object + channel (enum)
   Val_UnackAlmC : DINT; {access Read Only}   // Count of Unacknowledged Alarms
   Val_Owner : DINT; {access Read Only}   // Current Object Owner ID (0=not owned)
   Sts_St0 : BOOL; {access Read Only, visible}   // 1=Device commanded to and confirmed in State 0
   Sts_St1 : BOOL; {access Read Only, visible}   // 1=Device commanded to and confirmed in State 1
   Sts_St2 : BOOL; {access Read Only, visible}   // 1=Device commanded to and confirmed in State 2
   Sts_St3 : BOOL; {access Read Only, visible}   // 1=Device commanded to and confirmed in State 3
   Sts_Moving : BOOL; {access Read Only, visible}   // 1=Device not yet confirmed in commended state
   Sts_Horn : BOOL; {access Read Only}   // 1=Sound audible prior to commanded energize/ state change
   Sts_Available : BOOL; {access Read Only}   // 1=Device available for control by automation (Prog)
   Sts_Bypass : BOOL; {access Read Only}   // 1=Bypassable Interlocks and Permissives are Bypassed
   Sts_BypActive : BOOL; {access Read Only}   // 1=Interlock / Permissive Bypassing Active (Bypassed or Maintenance)
   Sts_NotRdy : BOOL; {access Read Only}   // 1=Device Not Ready, see detail bits for reason
   Nrdy_CfgErr : BOOL; {access Read Only}   // 1=Device Not Ready: Configuration Error
   Nrdy_EqpFault : BOOL; {access Read Only}   // 1=Device Not Ready: External Equipment Fault (Fault or Shed Requires Reset)
   Nrdy_Fail : BOOL; {access Read Only}   // 1=Device Not Ready: Device Failure (Shed Requires Reset)
   Nrdy_Intlk : BOOL; {access Read Only}   // 1=Device Not Ready: Interlock Not OK
   Nrdy_IOFault : BOOL; {access Read Only}   // 1=Device Not Ready: I/O Fault (Shed Requires Reset)
   Nrdy_OoS : BOOL; {access Read Only}   // 1=Device Not Ready: Device is Out of Service
   Nrdy_PrioSt0 : BOOL; {access Read Only}   // 1=Device Not Ready: Oper/Ext Priority State 0 Command Requires Reset
   Nrdy_Perm : BOOL; {access Read Only}   // 1=Device Not Ready: Permissive Not OK
   Sts_MaintByp : BOOL; {access Read Only}   // 1=Device has a Maintenance Bypass function active
   Sts_AlmInh : BOOL; {access Read Only}   // 1=One or more Alarms Shelved, Disabled or Suppressed
   Sts_Err : BOOL; {access Read Only, visible}   // 1=Error in Config: see detail bits for reason
   Err_Timer : BOOL; {access Read Only}   // 1=Error in Config: Feeback Check timer preset (use 0 to 2147483)
   Err_Sim : BOOL; {access Read Only}   // 1=Error in Config: Simulation timer preset (use 0 to 2147483)
   Err_Alarm : BOOL; {access Read Only}   // 1=Error in Config: Alarm Min On Time, Shelf Time, Severity
   Sts_Hand : ALIAS FOR CmdSrc.Sts_Hand; {access Read Only, visible}
   Sts_OoS : ALIAS FOR CmdSrc.Sts_OoS; {access Read Only, visible}
   Sts_Maint : ALIAS FOR CmdSrc.Sts_Maint; {access Read Only, visible}
   Sts_Ovrd : ALIAS FOR CmdSrc.Sts_Ovrd; {access Read Only, visible}
   Sts_Ext : ALIAS FOR CmdSrc.Sts_Ext; {access Read Only}
   Sts_Prog : ALIAS FOR CmdSrc.Sts_Prog; {access Read Only, visible}
   Sts_ProgLocked : ALIAS FOR CmdSrc.Sts_ProgLocked; {access Read Only, visible}
   Sts_Oper : ALIAS FOR CmdSrc.Sts_Oper; {access Read Only, visible}
   Sts_OperLocked : ALIAS FOR CmdSrc.Sts_OperLocked; {access Read Only, visible}
   Sts_Normal : ALIAS FOR CmdSrc.Sts_Normal; {access Read Only}
   Sts_ExtReqInh : ALIAS FOR CmdSrc.Sts_ExtReqInh; {access Read Only}
   Sts_ProgReqInh : ALIAS FOR CmdSrc.Sts_ProgReqInh; {access Read Only}
   Sts_MAcqRcvd : ALIAS FOR CmdSrc.Sts_MAcqRcvd; {access Read Only}
   Sts_RdyReset : ALIAS FOR ORdy_Reset; {access Read Only}   // 1=A latched alarm or shed condition is ready to be reset
   Sts_RdyAck : BOOL; {access Read Only}   // 1=An alarm is ready to be acknowledged
   Sts_Fail : ALIAS FOR Fail.Inp;   // 1=Device failed to reach commended state
   Alm_Fail : ALIAS FOR Fail.Alm;   // 1=Alarm: Device failed to reach commended state
   Ack_Fail : ALIAS FOR Fail.Ack;   // 1=Fail to reach commanded state Alarm has been acknowledged
   Sts_FailDisabled : ALIAS FOR Fail.Disabled;   // 1=Fail to reach commanded state Alarm has been Disabled by Maintenance
   Sts_FailShelved : ALIAS FOR Fail.Shelved;   // 1=Fail to reach commanded state Alarm has been Shelved by Operator
   Sts_FailSuppressed : ALIAS FOR Fail.Suppressed;   // 1=Fail to reach commanded state alarm has been Suppressed by Program
   Sts_DeviceFault : ALIAS FOR DeviceFault.Inp;   // 1=Device Fault (from Inp_DeviceFault)
   Alm_DeviceFault : ALIAS FOR DeviceFault.Alm;   // 1=Device Fault Alarm
   Ack_DeviceFault : ALIAS FOR DeviceFault.Ack;   // 1=Device Fault Alarm has been acknowledged
   Sts_DeviceFaultDisabled : ALIAS FOR DeviceFault.Disabled;   // 1=Device Fault Alarm has been Disabled by Maintenance
   Sts_DeviceFaultShelved : ALIAS FOR DeviceFault.Shelved;   // 1=Device Fault Alarm has been Shelved by Operator
   Sts_DeviceFaultSuppressed : ALIAS FOR DeviceFault.Suppressed;   // 1=Device Fault Alarm has been Suppressed by Program
   Sts_IntlkTrip : ALIAS FOR IntlkTrip.Inp;   // 1=Device commanded to State 0 by an Interlock NOT OK (one-shot)
   Alm_IntlkTrip : ALIAS FOR IntlkTrip.Alm;   // 1=Alarm: Device set to State 0 by an Interlock NOT OK
   Ack_IntlkTrip : ALIAS FOR IntlkTrip.Ack;   // 1=Interlock Trip Alarm has been acknowledged
   Sts_IntlkTripDisabled : ALIAS FOR IntlkTrip.Disabled;   // 1=Interlock Trip Alarm has been Disabled by Maintenance
   Sts_IntlkTripShelved : ALIAS FOR IntlkTrip.Shelved;   // 1=Interlock Trip Alarm has been Shelved by Operator
   Sts_IntlkTripSuppressed : ALIAS FOR IntlkTrip.Suppressed;   // 1=Interlock Trip Alarm has been Suppressed by Program
   Sts_IOFault : ALIAS FOR IOFault.Inp;   // I/O Comm Fault Status (0=OK, 1=Bad)
   Alm_IOFault : ALIAS FOR IOFault.Alm;   // 1=I/O Fault Alarm
   Ack_IOFault : ALIAS FOR IOFault.Ack;   // 1=I/O Fault Alarm has been acknowledged
   Sts_IOFaultDisabled : ALIAS FOR IOFault.Disabled;   // 1=I/O Fault Alarm has been Disabled by Maintenance
   Sts_IOFaultShelved : ALIAS FOR IOFault.Shelved;   // 1=I/O Fault Alarm has been Shelved by Operator
   Sts_IOFaultSuppressed : ALIAS FOR IOFault.Suppressed;   // 1=I/O Fault Alarm has been Suppressed by Program
   MRdy_Rel : ALIAS FOR CmdSrc.MRdy_Rel; {access Read Only}
   ORdy_Unlock : ALIAS FOR CmdSrc.ORdy_Unlock; {access Read Only}
   P_D4SD : BOOL;   // Unique Parameter Name for auto - discovery
END_VAR
VAR
   Wrk_OutDPulseT : TIMER; {access None}   // Output D Pulse Timer
   Wrk_OutCPulseT : TIMER; {access None}   // Output C Pulse Timer
   Wrk_OutBPulseT : TIMER; {access None}   // Output B Pulse Timer
   Wrk_OutAPulseT : TIMER; {access None}   // Output A Pulse Timer
   Wrk_Notify : DINT; {access None}   // Buffer for building Val_Notify
   Wrk_Bypass : BOOL; {access None}   // Internal Bypassable Permissives and Interlocks are Bypassed flag
   Wrk_ActState : DINT; {access None}   // Actual State (enum)
   Fail : P_Alarm := (Cfg_AckReqd := 1, Cfg_AllowShelve := 1, Cfg_AllowDisable := 1, Cfg_Severity := 1000, Cfg_AlmMinOnT := 5, PCfg_AllowExist := 1, Ack := 1);   // Device Fail to reach commanded position
   DeviceFault : P_Alarm := (Cfg_AckReqd := 1, Cfg_AllowShelve := 1, Cfg_AllowDisable := 1, Cfg_Severity := 1000, Cfg_AlmMinOnT := 5, PCfg_AllowExist := 1, Ack := 1);   // Device Fault from device via input
   CmdSrc : P_CmdSrc := (Cfg_HasOper := 1, Cfg_HasOperLocked := 1, Cfg_HasProg := 1, Cfg_HasProgLocked := 1, Cfg_HasMaint := 1, Cfg_HasMOoS := 1, Cfg_OvrdOverLock := 1, Sts_bSrc := 1, Sts_Oper := 1);   // Control / Command Source Selection
   IOFault : P_Alarm := (Cfg_AckReqd := 1, Cfg_AllowShelve := 1, Cfg_AllowDisable := 1, Cfg_Severity := 1000, Cfg_AlmMinOnT := 5, PCfg_AllowExist := 1, Ack := 1);   // I/O Fault Alarm
   IntlkTrip : P_Alarm := (Cfg_AckReqd := 1, Cfg_AllowShelve := 1, Cfg_AllowDisable := 1, Cfg_Severity := 500, Cfg_AlmMinOnT := 5, PCfg_AllowExist := 1, Ack := 1);   // Interlock Trip Alarm
   HMI_Tab : SINT;   // Tab to display (FTView ME)
   Wrk_ONS : SINT; {access None}   // One-Shot Store Bits
   Wrk_Out : SINT; {access None}   // Outputs (buffered) as a SINT for byte-wise operations
   Wrk_FdbkState : DINT; {access None}   // State(s) of device as shown by feedbacks
   Cfg_Tag : STRING_20 := 'P_D4SD';   // Tagname for display on HMI
   Cfg_Label : STRING_20 := 'Discrete Device';   // Label for graphic symbol displayed on HMI
   Cfg_Desc : STRING_40 := 'Discrete 2, 3 or 4 S';   // Description for display on HMI
   Cfg_St3Text : STRING_8;   // Text to display in State 3
   Cfg_St2Text : STRING_8;   // Text to display in State 2
   Cfg_St1Text : STRING_8 := 'On';   // Text to display in State 1
   Cfg_St0Text : STRING_8 := 'Off';   // Text to display in State 0
   Wrk_PermOK3 : BOOL; {access None}   // 1=Permissives are OK to go to state 3
   Wrk_PermOK2 : BOOL; {access None}   // 1=Permissives are OK to go to state 2
   Wrk_PermOK1 : BOOL; {access None}   // 1=Permissives are OK to go to state 1
   Wrk_PermOK0 : BOOL; {access None}   // 1=Permissives are OK to go to state 0
   Wrk_TgtState : DINT; {access None}   // Target device state as a number (0, 1, 2 or 3)
   Wrk_SimT : TIMER; {access None}   // Time "moving" before going to target pos. in simulation
   Wrk_FailT : TIMER; {access Read Only}   // Failure Check timer (time to reach target position)
   Wrk_NewCmd : BOOL; {access None}   // 1=A state command has been received (even for same state)
   Wrk_PrevTgt : DINT; {access None}   // Previous Target State (last scan)
   HMI_Type : STRING_16 := 'P_D4SD'; {access Read Only}   // Type identifier for HMI navigation
   HMI_Lib : STRING_12 := 'RA-BAS'; {access Read Only}   // Display Library for Faceplate call-up
   Wrk_Sts : DINT; {access None}   // Buffer for building Val_Sts
   Wrk_Fault : DINT; {access None}   // Buffer for building Val_Fault
   Wrk_SrcQ : DINT; {access None}   // Register for building Source / Quality enumeration
   Val_Notify : DINT; {access Read Only}   // Current Alarm Level and Acknowledgement (enumeration)
   Wrk_NotRdy : BOOL; {access None}   // Device Not Ready conditions excluding shed latches
   Wrk_NotRdy1 : BOOL; {access None}   // Device Not Ready excluding only Permissives
   Wrk_NoLongerSim : BOOL; {access None}   // Switched from Simulated to Real Device this scan
   Cfg_Area : STRING_Area := 'area01';   // Process Area for security
   Wrk_UnackAlmC : DINT; {access None}   // Buffer for building Val_UnackAlmC
   ORdy_ResetAckAll : BOOL; {access Read Only}   // 1=At least one Alarm or latched Shed requires Reset or Ack
   ORdy_Reset : BOOL; {access Read Only}   // 1=At least one Alarm or latched Shed requires Reset
   ORdy_St3 : BOOL; {access Read Only}   // 1=Ready for OCmd_St3, enable HMI button
   ORdy_St2 : BOOL; {access Read Only}   // 1=Ready for OCmd_St2, enable HMI button
   ORdy_St1 : BOOL; {access Read Only}   // 1=Ready for OCmd_St1, enable HMI button
   ORdy_St0 : BOOL; {access Read Only}   // 1=Ready for OCmd_St0, enable HMI button
   MRdy_Check : BOOL; {access Read Only}   // 1=Ready for MCmd_Check, enable HMI button
   MRdy_Bypass : BOOL; {access Read Only}   // 1=Ready for MCmd_Bypass, enable HMI button
   OCmd_ResetAckAll : BOOL;   // Oper Cmd to reset shed latches and cleared alarms, plus Acknowledge alarms
   OCmd_Reset : BOOL;   // Oper Cmd to reset shed latches and cleared alarms
   OCmd_St3 : BOOL;   // Operator Command to set device to State 3
   OCmd_St2 : BOOL;   // Operator Command to set device to State 2
   OCmd_St1 : BOOL;   // Operator Command to set device to State 1
   OCmd_St0 : BOOL;   // Operator Command to set device to State 0
   MCmd_Check : BOOL;   // Maintenance Command to Check Interlocks and Permissives
   MCmd_Bypass : BOOL;   // Maintenance Command to Bypass Interlocks and Permissives
   Wrk_StartHornT : TIMER; {access None}   // Timer for audible alert or start
   Wrk_StartHorn : BOOL; {access None}   // 1=Sound audible prior to commanded energize/ state change
   Wrk_TgtStateTmp : DINT; {access None}   // Target device state as a number (0, 1, 2 or 3) stored, before audible alert
   Wrk_AfterHornONS : BOOL; {access None}
   Wrk_AfterHornONS2 : BOOL; {access None}
END_VAR

ROUTINE EnableInFalse   (* ladder *)
// Out of Service is asserted; Outputs OFF; Device Status shown based on feedbacks if possible, but Alarms inhibited
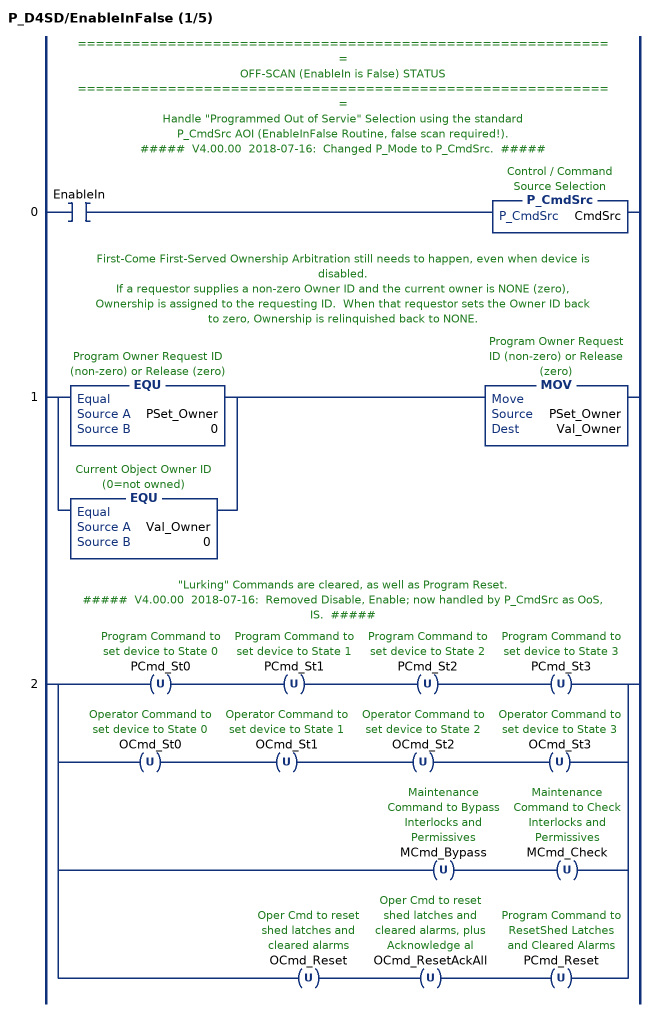
   // ============================================================
   // OFF-SCAN (EnableIn is False) STATUS
   // ============================================================
   // Handle "Programmed Out of Servie" Selection using the standard
   // P_CmdSrc AOI (EnableInFalse Routine, false scan required!).
   // #####  V4.00.00  2018-07-16:  Changed P_Mode to P_CmdSrc.  #####
   0: XIC(EnableIn)P_CmdSrc(CmdSrc);
   // First-Come First-Served Ownership Arbitration still needs to happen, even when device is disabled.
   // If a requestor supplies a non-zero Owner ID and the current owner is NONE (zero),
   // Ownership is assigned to the requesting ID.  When that requestor sets the Owner ID back
   // to zero, Ownership is relinquished back to NONE.
   1: [EQU(PSet_Owner,0) ,EQU(Val_Owner,0) ]MOV(PSet_Owner,Val_Owner);
   // "Lurking" Commands are cleared, as well as Program Reset.
   // #####  V4.00.00  2018-07-16:  Removed Disable, Enable; now handled by P_CmdSrc as OoS, IS.  #####
   2: [OTU(PCmd_St0) OTU(PCmd_St1) OTU(PCmd_St2) OTU(PCmd_St3) ,OTU(OCmd_St0) OTU(OCmd_St1) OTU(OCmd_St2) OTU(OCmd_St3) ,OTU(MCmd_Bypass) OTU(MCmd_Check) ,OTU(OCmd_Reset) OTU(OCmd_ResetAckAll) OTU(PCmd_Reset) ];
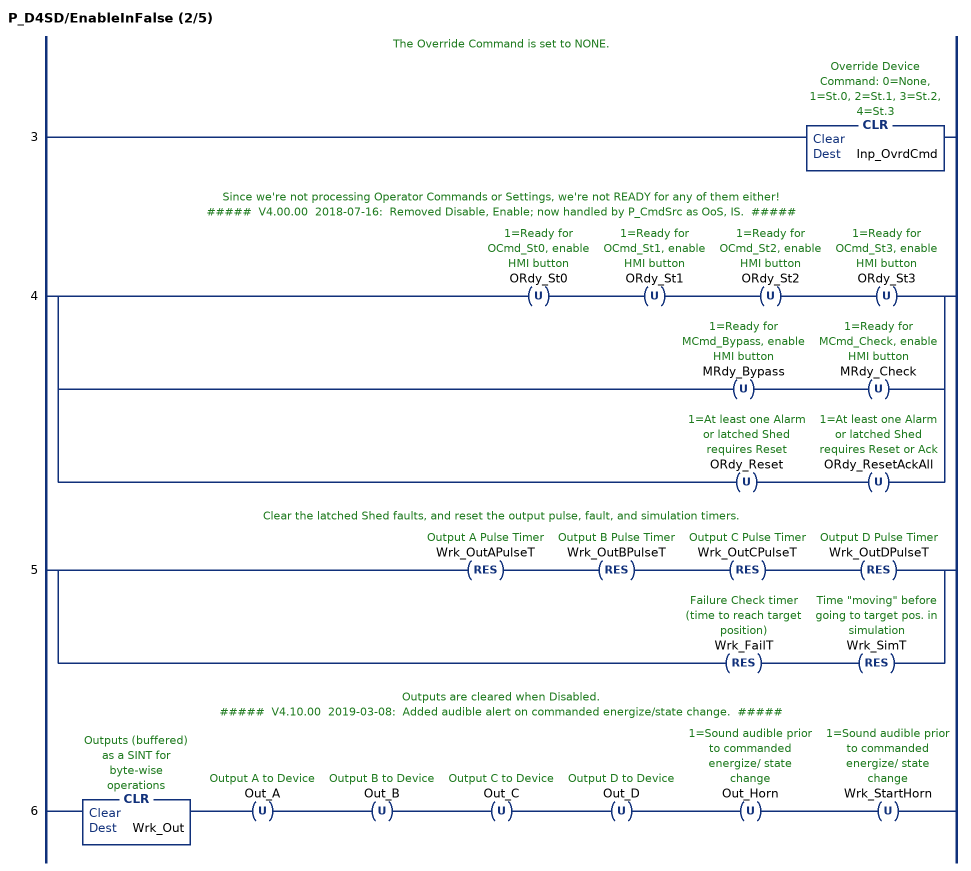
   // The Override Command is set to NONE.
   3: CLR(Inp_OvrdCmd);
   // Since we're not processing Operator Commands or Settings, we're not READY for any of them either!
   // #####  V4.00.00  2018-07-16:  Removed Disable, Enable; now handled by P_CmdSrc as OoS, IS.  #####
   4: [OTU(ORdy_St0) OTU(ORdy_St1) OTU(ORdy_St2) OTU(ORdy_St3) ,OTU(MRdy_Bypass) OTU(MRdy_Check) ,OTU(ORdy_Reset) OTU(ORdy_ResetAckAll) ];
   // Clear the latched Shed faults, and reset the output pulse, fault, and simulation timers.
   5: [RES(Wrk_OutAPulseT) RES(Wrk_OutBPulseT) RES(Wrk_OutCPulseT) RES(Wrk_OutDPulseT) ,RES(Wrk_FailT) RES(Wrk_SimT) ];
   // Outputs are cleared when Disabled.
   // #####  V4.10.00  2019-03-08:  Added audible alert on commanded energize/state change.  #####
   6: CLR(Wrk_Out)OTU(Out_A)OTU(Out_B)OTU(Out_C)OTU(Out_D)OTU(Out_Horn)OTU(Wrk_StartHorn);
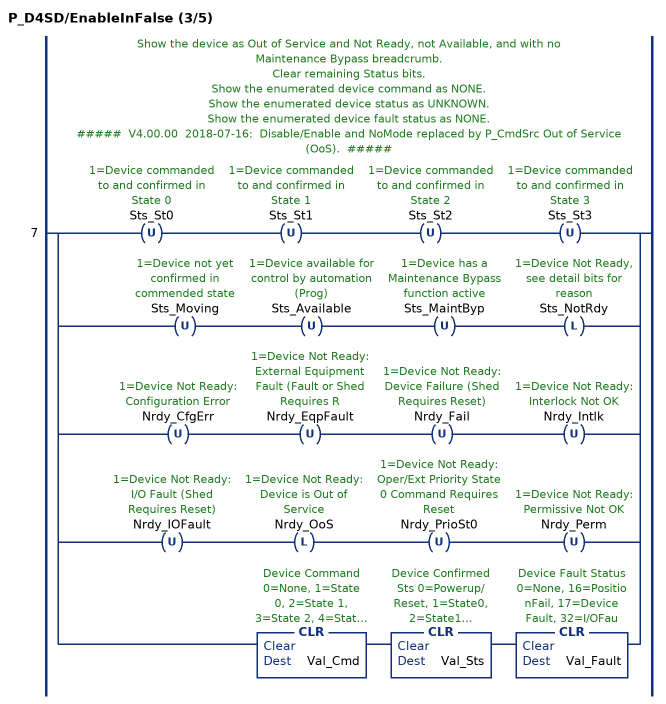
   // Show the device as Out of Service and Not Ready, not Available, and with no
   // Maintenance Bypass breadcrumb.
   // Clear remaining Status bits.
   // Show the enumerated device command as NONE.
   // Show the enumerated device status as UNKNOWN.
   // Show the enumerated device fault status as NONE.
   // #####  V4.00.00  2018-07-16:  Disable/Enable and NoMode replaced by P_CmdSrc Out of Service (OoS).  #####
   7: [OTU(Sts_St0) OTU(Sts_St1) OTU(Sts_St2) OTU(Sts_St3) ,OTU(Sts_Moving) OTU(Sts_Available) OTU(Sts_MaintByp) OTL(Sts_NotRdy) ,OTU(Nrdy_CfgErr) OTU(Nrdy_EqpFault) OTU(Nrdy_Fail) OTU(Nrdy_Intlk) ,OTU(Nrdy_IOFault) OTL(Nrdy_OoS) OTU(Nrdy_PrioSt0) OTU(Nrdy_Perm) ,CLR(Val_Cmd) CLR(Val_Sts) CLR(Val_Fault) ];
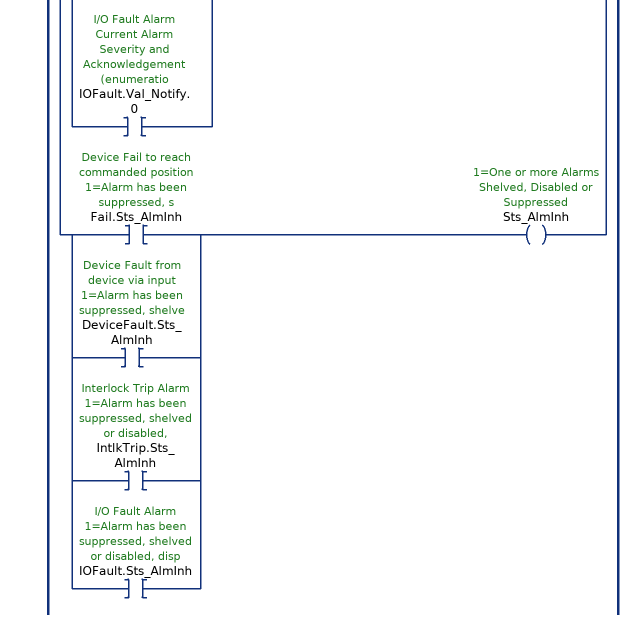
   // If the device is OFF-SCAN (rung is false or EnableIn is false in FBD),
   // then show the alarms as "Parent object out of service".
   // Show the overall acknowledgement status.
   // #####  V4.00.00  2018-07-16:  Changed P_Mode to P_CmdSrc, added Out of Service.  #####
   8: [OTL(Fail.Inp_OoS) P_Alarm(Fail) ,OTL(DeviceFault.Inp_OoS) P_Alarm(DeviceFault) ,OTL(IntlkTrip.Inp_OoS) P_Alarm(IntlkTrip) ,OTL(IOFault.Inp_OoS) P_Alarm(IOFault) ,CLR(Val_Notify) CLR(Val_NotifyAll) ,[XIC(Fail.Val_Notify.0) ,XIC(DeviceFault.Val_Notify.0) ,XIC(IntlkTrip.Val_Notify.0) ,XIC(IOFault.Val_Notify.0) ] OTL(Val_Notify.0) OTL(Val_NotifyAll.0) ,[XIC(Fail.Sts_AlmInh) ,XIC(DeviceFault.Sts_AlmInh) ,XIC(IntlkTrip.Sts_AlmInh) ,XIC(IOFault.Sts_AlmInh) ] OTE(Sts_AlmInh) ];
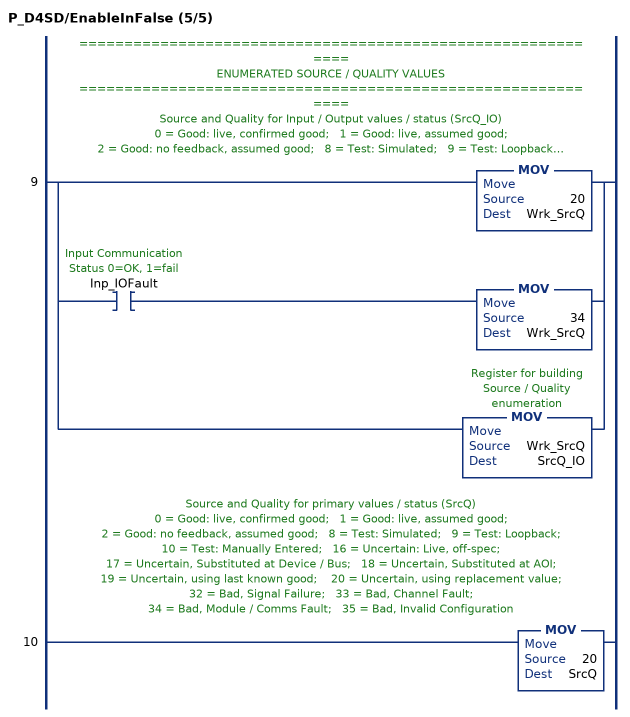
   // ============================================================
   // ENUMERATED SOURCE / QUALITY VALUES
   // ============================================================
   // Source and Quality for Input / Output values / status (SrcQ_IO)
   // 0 = Good: live, confirmed good;   1 = Good: live, assumed good;
   // 2 = Good: no feedback, assumed good;   8 = Test: Simulated;   9 = Test: Loopback;
   // 10 = Test: Manually Entered;   16 = Uncertain: Live, off-spec;
   // 17 = Uncertain, Substituted at Device / Bus;   18 = Uncertain, Substituted at AOI;
   // 19 = Uncertain, using last known good;    20 = Uncertain, using replacement value;
   // 32 = Bad, Signal Failure;   33 = Bad, Channel Fault;
   // 34 = Bad, Module / Comms Fault;   35 = Bad, Invalid Configuration
   9: [MOV(20,Wrk_SrcQ) ,XIC(Inp_IOFault) MOV(34,Wrk_SrcQ) ,MOV(Wrk_SrcQ,SrcQ_IO) ];
   // Source and Quality for primary values / status (SrcQ)
   // 0 = Good: live, confirmed good;   1 = Good: live, assumed good;
   // 2 = Good: no feedback, assumed good;   8 = Test: Simulated;   9 = Test: Loopback;
   // 10 = Test: Manually Entered;   16 = Uncertain: Live, off-spec;
   // 17 = Uncertain, Substituted at Device / Bus;   18 = Uncertain, Substituted at AOI;
   // 19 = Uncertain, using last known good;    20 = Uncertain, using replacement value;
   // 32 = Bad, Signal Failure;   33 = Bad, Channel Fault;
   // 34 = Bad, Module / Comms Fault;   35 = Bad, Invalid Configuration
   10: MOV(20,SrcQ);
END_ROUTINE
